// TIA Portal V17 export
// export: Created 2023-02-14T02:49:23.0844074Z, ExportSetting WithDefaults, DisplayName Totally Integrated Automation Portal, DisplayVersion V17, DisplayName TIA Portal Openness, DisplayVersion V17, DisplayName TIA Portal Teamcenter Gateway, DisplayVersion V17, DisplayName TIA Portal Version Control Interface, DisplayVersion V17, DisplayName SINAMICS Startdrive Advanced, DisplayVersion V17, DisplayName SINAMICS Startdrive G130, G150, S120, S150, SINAMICS MV, S210, DisplayVersion V17, DisplayName SINAMICS Startdrive G110M, G120, G120C, G120D, G120P, G115D, DisplayVersion V17, DisplayName STEP 7 Professional, DisplayVersion V17, DisplayName STEP 7 Safety, DisplayVersion V17, DisplayName WinCC Professional, DisplayVersion V17
FUNCTION_BLOCK "IO Digital Homomixer"   // FB5, LAD
{ S7_Optimized_Access := 'FALSE' }
VERSION : 0.1
// stored: AutoNumber true, IsIECCheckEnabled false, SetENOAutomatically false, UDAEnableTagReadback false
   VAR_INPUT
      Init : Bool;
      Reset : Bool;
   END_VAR
   VAR
      "LL-12.01" { S7_SetPoint := 'True'} : "Digital";   // LOW LEVEL SENSOR HOMOMIXER T-12.00
      "LL-13.01" { S7_SetPoint := 'True'} : "Digital";   // LOW LEVEL SENSOR HOMOMIXER T-13.00
      "LL-14.01" { S7_SetPoint := 'True'} : "Digital";
   END_VAR
BEGIN

REGION Network 1: LL-12.01 LOW LEVEL SENSOR HOMOMIXER T-12.00
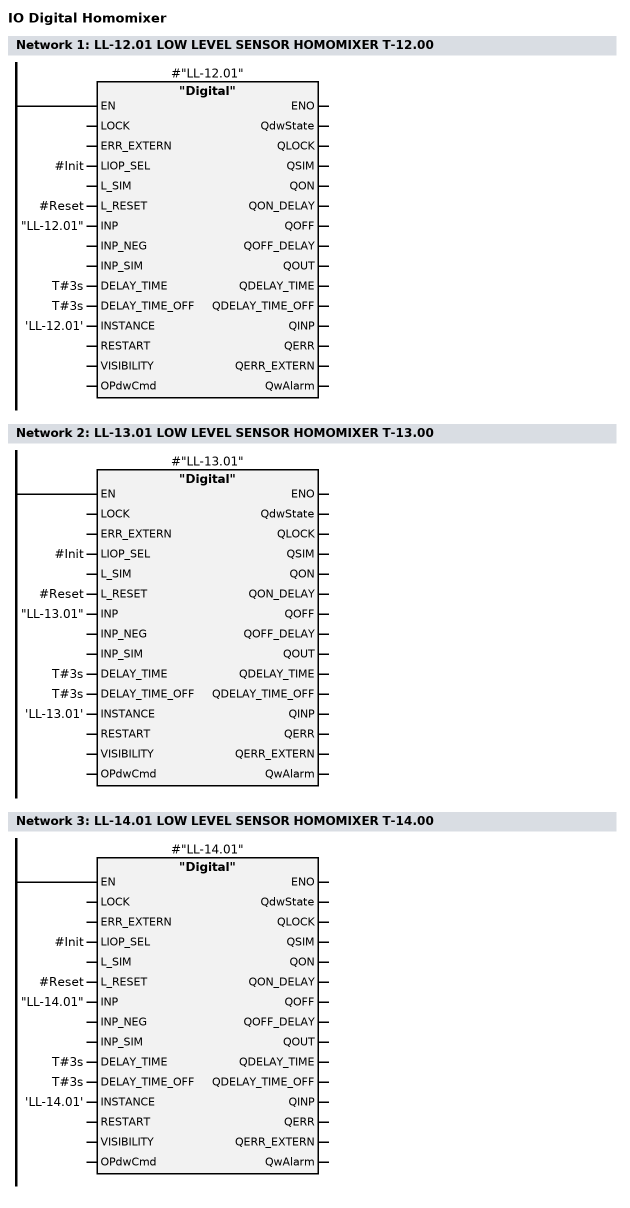
   RUNG wire#powerrail
      #"LL-12.01"(LOCK :=, ERR_EXTERN :=, LIOP_SEL := #Init, L_SIM :=, L_RESET := #Reset, INP := "LL-12.01", INP_NEG :=, INP_SIM :=, DELAY_TIME := T#3s, DELAY_TIME_OFF := T#3s, INSTANCE := 'LL-12.01', RESTART :=, VISIBILITY :=, OPdwCmd :=, QdwState =>, QLOCK =>, QSIM =>, QON =>, QON_DELAY =>, QOFF =>, QOFF_DELAY =>, QOUT =>, QDELAY_TIME =>, QDELAY_TIME_OFF =>, QINP =>, QERR =>, QERR_EXTERN =>, QwAlarm =>)
   END_RUNG
   // the same network as SCL:
   #"LL-12.01"(LIOP_SEL := #Init,   // "Digital"
               L_RESET := #Reset,
               INP := "LL-12.01",
               DELAY_TIME := T#3s,
               DELAY_TIME_OFF := T#3s,
               INSTANCE := 'LL-12.01');
END_REGION

REGION Network 2: LL-13.01 LOW LEVEL SENSOR HOMOMIXER T-13.00
   RUNG wire#powerrail
      #"LL-13.01"(LOCK :=, ERR_EXTERN :=, LIOP_SEL := #Init, L_SIM :=, L_RESET := #Reset, INP := "LL-13.01", INP_NEG :=, INP_SIM :=, DELAY_TIME := T#3s, DELAY_TIME_OFF := T#3s, INSTANCE := 'LL-13.01', RESTART :=, VISIBILITY :=, OPdwCmd :=, QdwState =>, QLOCK =>, QSIM =>, QON =>, QON_DELAY =>, QOFF =>, QOFF_DELAY =>, QOUT =>, QDELAY_TIME =>, QDELAY_TIME_OFF =>, QINP =>, QERR =>, QERR_EXTERN =>, QwAlarm =>)
   END_RUNG
   // the same network as SCL:
   #"LL-13.01"(LIOP_SEL := #Init,   // "Digital"
               L_RESET := #Reset,
               INP := "LL-13.01",
               DELAY_TIME := T#3s,
               DELAY_TIME_OFF := T#3s,
               INSTANCE := 'LL-13.01');
END_REGION

REGION Network 3: LL-14.01 LOW LEVEL SENSOR HOMOMIXER T-14.00
   RUNG wire#powerrail
      #"LL-14.01"(LOCK :=, ERR_EXTERN :=, LIOP_SEL := #Init, L_SIM :=, L_RESET := #Reset, INP := "LL-14.01", INP_NEG :=, INP_SIM :=, DELAY_TIME := T#3s, DELAY_TIME_OFF := T#3s, INSTANCE := 'LL-14.01', RESTART :=, VISIBILITY :=, OPdwCmd :=, QdwState =>, QLOCK =>, QSIM =>, QON =>, QON_DELAY =>, QOFF =>, QOFF_DELAY =>, QOUT =>, QDELAY_TIME =>, QDELAY_TIME_OFF =>, QINP =>, QERR =>, QERR_EXTERN =>, QwAlarm =>)
   END_RUNG
   // the same network as SCL:
   #"LL-14.01"(LIOP_SEL := #Init,   // "Digital"
               L_RESET := #Reset,
               INP := "LL-14.01",
               DELAY_TIME := T#3s,
               DELAY_TIME_OFF := T#3s,
               INSTANCE := 'LL-14.01');
END_REGION
END_FUNCTION_BLOCK
